Universal Robots PolyScope program: d_full_bow.urp

Program d_full_bow (installation=string_planes directory=/programs/strings createdIn=5.17.3 lastSavedIn=5.17.3 robotSerialNumber=20245501435)
Calibrated DH parameters: a=[0.000154, -0.137004, -0.385524, -0.00002, 0.000092, 0]; d=[0.162441, 211.794786, -230.585024, 18.923638, 0.099786, 0.09951]; alpha=[1.569493, -0.001902, 0.003874, 1.570111, -1.570167, 0]; deltaTheta=[0, -1.242934, 1.056292, 0.186646, 0.000002, 0.000001]
InitVariablesNode
Robot Program (runOnlyOnce=false)
  MoveL speed 250 mm/s, acceleration 1200 mm/s^2 (useActiveTCP=true) feature=Base
    Waypoint Waypoint_1: TCP in base x=354.162 y=752.956 z=112.35 mm, rx=-1.4072 ry=-1.8657 rz=1.1589 rad; joints [-128.358, -13.678, 35.826, -55.435, -63.826, -158.494] deg; TCP offset x=28.21 y=-96.107 z=-99.69 mm, rx=0 ry=0 rz=0 rad
    Waypoint Waypoint_3: TCP in base x=382.369 y=223.018 z=171.533 mm, rx=-1.5103 ry=-1.95 rz=1.0441 rad; joints [-170.953, -57.66, 119.157, -99.41, -99.245, -180.678] deg
  SuppressedNode
    MoveL speed 250 mm/s, acceleration 1200 mm/s^2 (useActiveTCP=true) feature=Base
      Waypoint Waypoint_3: TCP in base x=447.609 y=273.936 z=153.016 mm, rx=-1.5094 ry=-2.0788 rz=1.1993 rad; joints [-166.924, -49.251, 104.272, -93.996, -106.227, -176.948] deg
      Waypoint Waypoint_1: TCP in base x=358.556 y=758.659 z=94.067 mm, rx=-1.5094 ry=-2.0788 rz=1.1993 rad; joints [-129.115, -10.524, 30.67, -58.491, -76.391, -153.642] deg
  Wait Sleep waitTime=300
  bow_dir := True
  note_dur := 1
  Timer (action=Start) variable(name=timer_1)
  If bow_dir≟ False
    MoveL speed 250 mm/s, acceleration 1200 mm/s^2 (useActiveTCP=true) feature=Base
      Waypoint Waypoint_1: TCP in base x=354.162 y=752.956 z=112.35 mm, rx=-1.4072 ry=-1.8657 rz=1.1589 rad; joints [-128.358, -13.678, 35.826, -55.435, -63.826, -158.494] deg
        Until EXPRESSION (allowActions=false) ExpressionBranch=timer_1≟note_dur
  Else 
    MoveL speed 250 mm/s, acceleration 1200 mm/s^2 (useActiveTCP=true) feature=Base
      Waypoint Waypoint_3: TCP in base x=382.369 y=223.018 z=171.533 mm, rx=-1.5103 ry=-1.95 rz=1.0441 rad; joints [-170.953, -57.66, 119.157, -99.41, -99.245, -180.678] deg
        Until EXPRESSION (allowActions=false) ExpressionBranch=timer_1≟note_dur
  SuppressedNode
    MoveL speed 250 mm/s, acceleration 1200 mm/s^2 (useActiveTCP=true) feature=Base
      Waypoint Waypoint_1: TCP in base x=331.973 y=720.894 z=108.291 mm, rx=-1.645 ry=-2.1081 rz=1.0591 rad; joints [-129.773, -21.651, 52.373, -76.468, -76.907, -149.022] deg
      Waypoint Waypoint_2: motionParameters(blendRadius=0.05); TCP in base x=332.259 y=481.199 z=108.291 mm, rx=-1.645 ry=-2.1081 rz=1.0591 rad; joints [-144.031, -41.816, 97.865, -100.392, -86.961, -159.136] deg
      Waypoint Waypoint_3: TCP in base x=332.566 y=223.853 z=108.291 mm, rx=-1.645 ry=-2.1081 rz=1.0591 rad; joints [-170.229, -51.627, 126.122, -120.942, -105.516, -177.767] deg
  Timer (action=Stop) variable=timer_1
  Timer (action=Reset) variable=timer_1
